Omron CX-Programmer project НовыйПроект (CX-Programmer 9.61)

# PLC НовыйПЛК1: CP1E N30

## Global symbols (name address type ; comment)
0.00 BOOL  ; Pulsador 00. Control valvula 00, easy box 1.
0.01 BOOL  ; Pulsadoe 01_control valvula 01. Easy box 2.
0.02 BOOL  ; Pulsador 02, activa valvula 02 y bomba B00_B01 en alternancia.
0.03 BOOL  ; Pulsador03, activa valvula 03.
0.04 BOOL  ; Pulsador 04, activa valvula 04 y G.Presion B00_B01.
0.05 BOOL  ; Pulsador05, activa valvula 05 y G.presion B00_B01.
100.00 BOOL  ; Valvula V00
100.01 BOOL  ; Valvula V01
100.02 BOOL  ; Valvula V02.
100.03 BOOL  ; Valvula V03.
100.04 BOOL  ; Valvula V04.
100.05 BOOL  ; Valvula V05.
101.00 BOOL  ; Bomba B00.
101.01 BOOL  ; Bomba B01.
101.02 BOOL  ; Bomba Filtracion f01
101.03 BOOL  ; Bomba Filtracion f02
1.00 BOOL  ; Guardamotor B00.
1.01 BOOL  ; Guardamotor B01.
1.02 BOOL  ; Guardamotor filtraciуn.
1.03 BOOL  ; Reloj_termostato filtracion.
D0 CHANNEL  ; D.M Valor activar bomba B00
D1 CHANNEL  ; D.M Valor temporizacion B00
D10 CHANNEL  ; D.M Valor activar bomba B01
D11 CHANNEL  ; D.M valor temporizacion B01
T000 BOOL  ; Retardo V02 arranque bomba B00_B01,
T001 BOOL  ; Retardo V02 arranque bomba B00_B01,
T002 BOOL  ; Retardo V02 arranque bomba B00_B01,
T003 BOOL  ; Retardo V03 arranque bomba B00_B01,
T004 BOOL  ; Retardo V04 arranque bomba B00_B01,
T005 BOOL  ; Retardo V05 arranque bomba B00_B01,
W0.00 BOOL  ; Trabajo pulsador 00_valvula 00
W0.01 BOOL  ; Trabajo pulsador 00_valvula00
W0.02 BOOL  ; Salida Virtual valvula00
W0.05 BOOL  ; Trabajo Pulsador01_valvula01
W0.06 BOOL  ; Trabajo pulsador01_valvula01.
W0.07 BOOL  ; Salida Virtual valvula 01.
W0.10 BOOL  ; Trabajo pulsador02_valvula02
W0.11 BOOL  ; Trabajo pulsador02_valvula02
W0.12 BOOL  ; Salida virtual valvula02
W100 CHANNEL  ; Temporal valor bomba B00
W100.00 BOOL  ; Salida virtual Bomba B00
W100.01 BOOL  ; Salida virtual bomba B01
W100.10 BOOL  ; Salida virtual filtraciуn.
W101 CHANNEL  ; Temporal bomba B01
W101.01 BOOL  ; Virtual bomba B01
W1.00 BOOL  ; Trabajo pulsador03_valvula03.
W1.01 BOOL  ; Trabajo pulsador03_valvula03
W1.02 BOOL  ; Salida virtual valvula03
W1.05 BOOL  ; Trabajo pulsador04_valvula04
W1.06 BOOL  ; Trabajo pulsador04_valvula04
W1.07 BOOL  ; Salida virtual valvula04
W1.10 BOOL  ; Trabajo pulsador 05_valvula05
W1.11 BOOL  ; Trabajo pulsador05_valvula05
W1.12 BOOL  ; Salida virtual valvula05
W20.00 BOOL  ; Salida virtual valvula 00
W20.01 BOOL  ; Salida virtual valvula 01
W20.02 BOOL  ; Salida virtual valvula 02
W20.03 BOOL  ; Salida virtual valvula 03
W20.04 BOOL  ; Salida virtual valvula 04
W20.05 BOOL  ; Salida virtual valvula 05
W20.10 BOOL  ; Виртуальна переменная для ыключения насоса 01
W20.11 BOOL  ; Виртуальна переменная для ыключения насоса 02
W30.00 BOOL  ; Salida virtual valvula02
W30.02 BOOL  ; Seсal V02 arranque B00_B01.
W50 CHANNEL  ; Registro incremento temporizacion alternancia

## Program NuevoPrograma1 (cyclic task 0)
Local symbols
do CHANNEL

### Section Enclavamiento_pulsadores

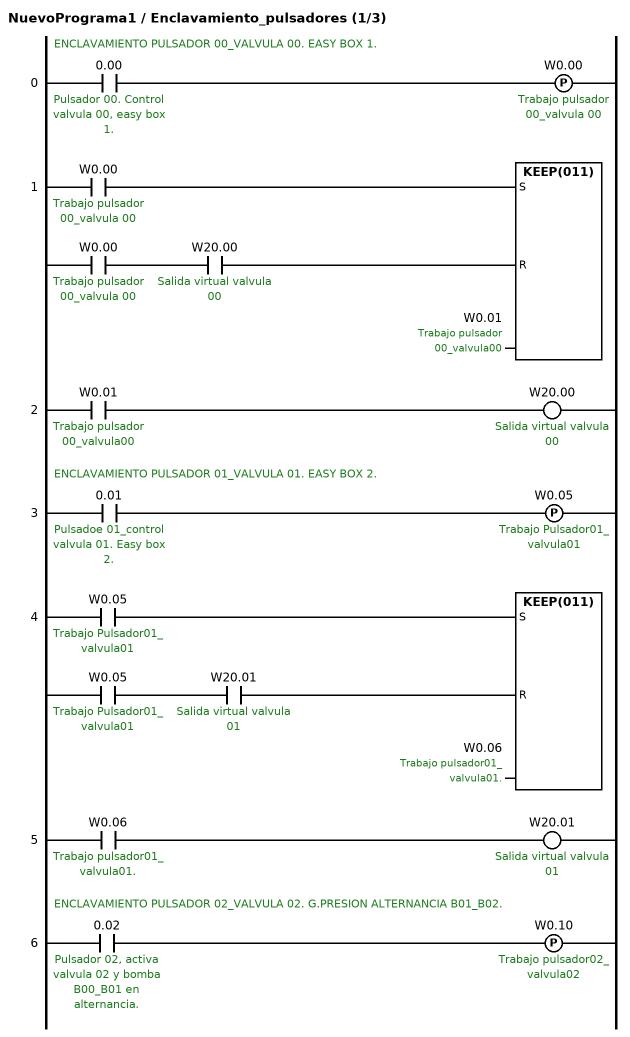
; rung 0: ENCLAVAMIENTO PULSADOR 00_VALVULA 00. EASY BOX 1.
LD 0.00  ; Pulsador 00. Control valvula 00, easy box 1.
DIFU(013) W0.00  ; Trabajo pulsador 00_valvula 00
; rung 1
LD W0.00  ; Trabajo pulsador 00_valvula 00
LD W0.00  ; Trabajo pulsador 00_valvula 00
AND W20.00  ; Salida virtual valvula 00
KEEP(011) W0.01  ; Trabajo pulsador 00_valvula00
; rung 2
LD W0.01  ; Trabajo pulsador 00_valvula00
OUT W20.00  ; Salida virtual valvula 00
; rung 3: ENCLAVAMIENTO PULSADOR 01_VALVULA 01. EASY BOX 2.
LD 0.01  ; Pulsadoe 01_control valvula 01. Easy box 2.
DIFU(013) W0.05  ; Trabajo Pulsador01_valvula01
; rung 4
LD W0.05  ; Trabajo Pulsador01_valvula01
LD W0.05  ; Trabajo Pulsador01_valvula01
AND W20.01  ; Salida virtual valvula 01
KEEP(011) W0.06  ; Trabajo pulsador01_valvula01.
; rung 5
LD W0.06  ; Trabajo pulsador01_valvula01.
OUT W20.01  ; Salida virtual valvula 01
; rung 6: ENCLAVAMIENTO PULSADOR 02_VALVULA 02. G.PRESION ALTERNANCIA B01_B02.
LD 0.02  ; Pulsador 02, activa valvula 02 y bomba B00_B01 en alternancia.
DIFU(013) W0.10  ; Trabajo pulsador02_valvula02

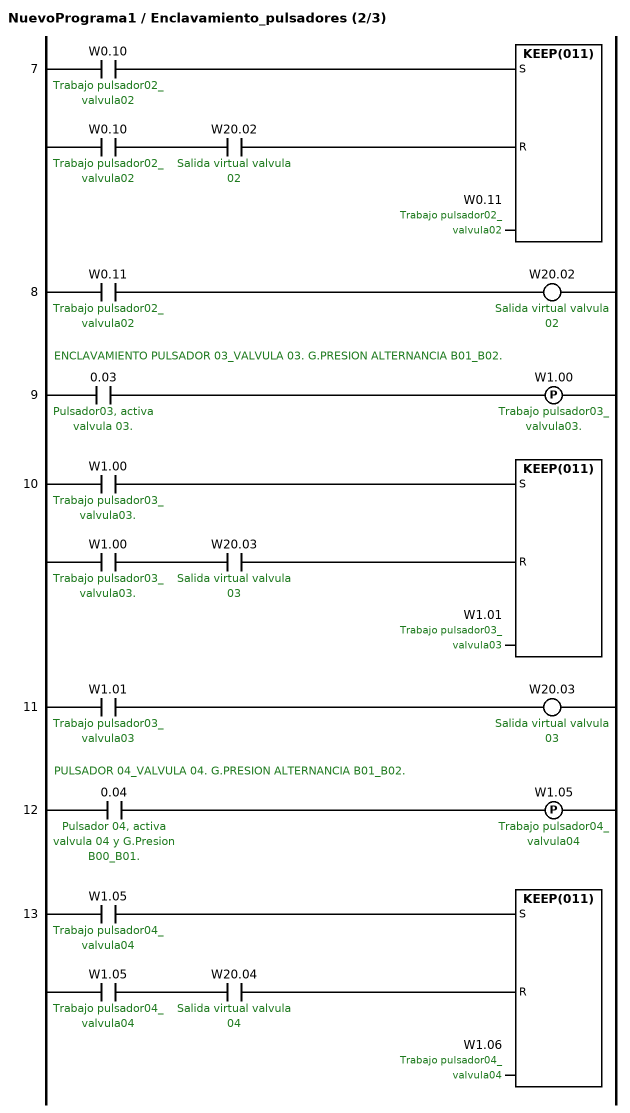
; rung 7
LD W0.10  ; Trabajo pulsador02_valvula02
LD W0.10  ; Trabajo pulsador02_valvula02
AND W20.02  ; Salida virtual valvula 02
KEEP(011) W0.11  ; Trabajo pulsador02_valvula02
; rung 8
LD W0.11  ; Trabajo pulsador02_valvula02
OUT W20.02  ; Salida virtual valvula 02
; rung 9: ENCLAVAMIENTO PULSADOR 03_VALVULA 03. G.PRESION ALTERNANCIA B01_B02.
LD 0.03  ; Pulsador03, activa valvula 03.
DIFU(013) W1.00  ; Trabajo pulsador03_valvula03.
; rung 10
LD W1.00  ; Trabajo pulsador03_valvula03.
LD W1.00  ; Trabajo pulsador03_valvula03.
AND W20.03  ; Salida virtual valvula 03
KEEP(011) W1.01  ; Trabajo pulsador03_valvula03
; rung 11
LD W1.01  ; Trabajo pulsador03_valvula03
OUT W20.03  ; Salida virtual valvula 03
; rung 12: PULSADOR 04_VALVULA 04. G.PRESION ALTERNANCIA B01_B02.
LD 0.04  ; Pulsador 04, activa valvula 04 y G.Presion B00_B01.
DIFU(013) W1.05  ; Trabajo pulsador04_valvula04
; rung 13
LD W1.05  ; Trabajo pulsador04_valvula04
LD W1.05  ; Trabajo pulsador04_valvula04
AND W20.04  ; Salida virtual valvula 04
KEEP(011) W1.06  ; Trabajo pulsador04_valvula04

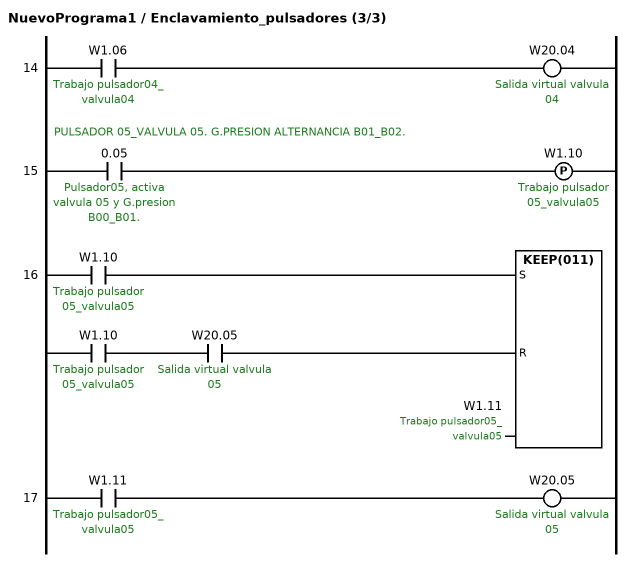
; rung 14
LD W1.06  ; Trabajo pulsador04_valvula04
OUT W20.04  ; Salida virtual valvula 04
; rung 15: PULSADOR 05_VALVULA 05. G.PRESION ALTERNANCIA B01_B02.
LD 0.05  ; Pulsador05, activa valvula 05 y G.presion B00_B01.
DIFU(013) W1.10  ; Trabajo pulsador 05_valvula05
; rung 16
LD W1.10  ; Trabajo pulsador 05_valvula05
LD W1.10  ; Trabajo pulsador 05_valvula05
AND W20.05  ; Salida virtual valvula 05
KEEP(011) W1.11  ; Trabajo pulsador05_valvula05
; rung 17
LD W1.11  ; Trabajo pulsador05_valvula05
OUT W20.05  ; Salida virtual valvula 05

### Section Alternancia_bombas_B00_B01

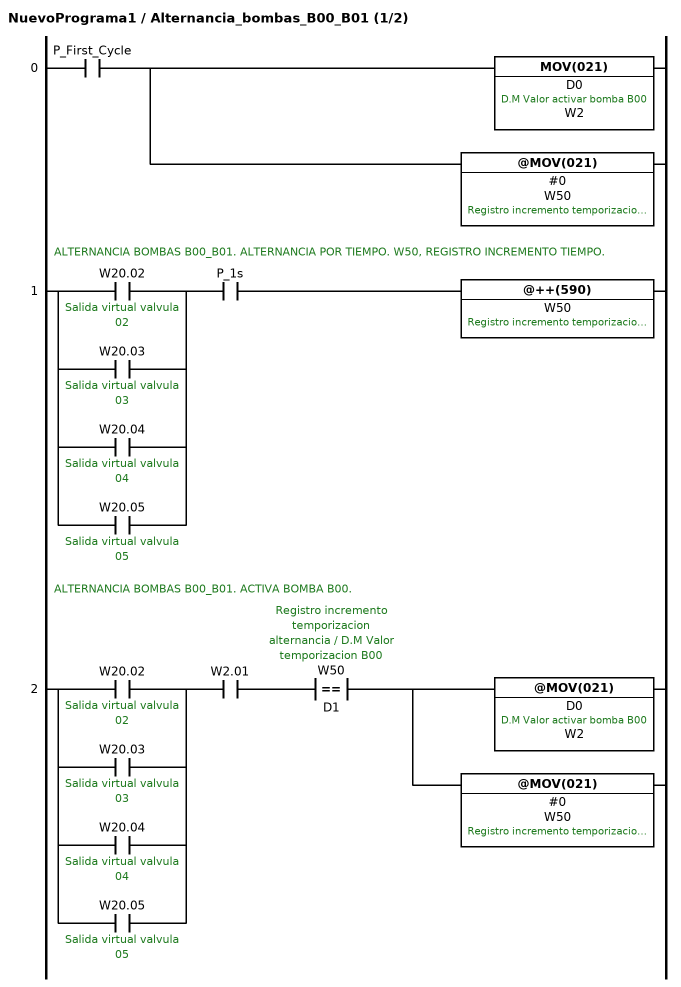
; rung 0
LD P_First_Cycle
MOV(021) D0 W2  ; D.M Valor activar bomba B00
@MOV(021) #0 W50  ; Registro incremento temporizacion alternancia
; rung 1: ALTERNANCIA BOMBAS B00_B01. ALTERNANCIA POR TIEMPO. W50, REGISTRO INCREMENTO TIEMPO.
LD W20.02  ; Salida virtual valvula 02
OR W20.03  ; Salida virtual valvula 03
OR W20.04  ; Salida virtual valvula 04
OR W20.05  ; Salida virtual valvula 05
AND P_1s
@++(590) W50  ; Registro incremento temporizacion alternancia
; rung 2: ALTERNANCIA BOMBAS B00_B01. ACTIVA BOMBA B00.
LD W20.02  ; Salida virtual valvula 02
OR W20.03  ; Salida virtual valvula 03
OR W20.04  ; Salida virtual valvula 04
OR W20.05  ; Salida virtual valvula 05
AND W2.01
AND=(300) W50 D1  ; Registro incremento temporizacion alternancia, D.M Valor temporizacion B00
@MOV(021) D0 W2  ; D.M Valor activar bomba B00
@MOV(021) #0 W50  ; Registro incremento temporizacion alternancia

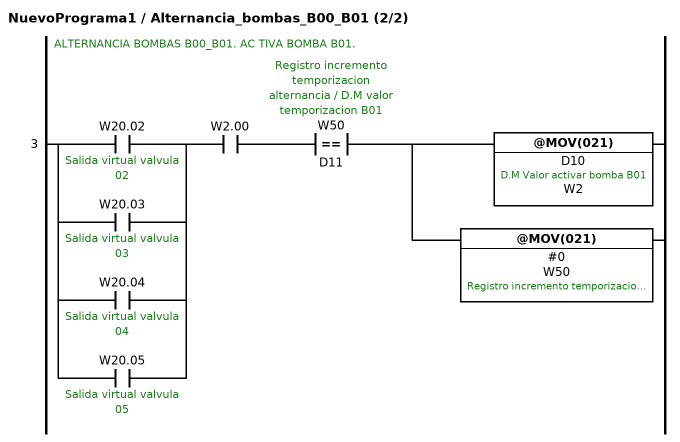
; rung 3: ALTERNANCIA BOMBAS B00_B01. AC TIVA BOMBA B01.
LD W20.02  ; Salida virtual valvula 02
OR W20.03  ; Salida virtual valvula 03
OR W20.04  ; Salida virtual valvula 04
OR W20.05  ; Salida virtual valvula 05
AND W2.00
AND=(300) W50 D11  ; Registro incremento temporizacion alternancia, D.M valor temporizacion B01
@MOV(021) D10 W2  ; D.M Valor activar bomba B01
@MOV(021) #0 W50  ; Registro incremento temporizacion alternancia

### Section Retardos_arranque_bombas00_01

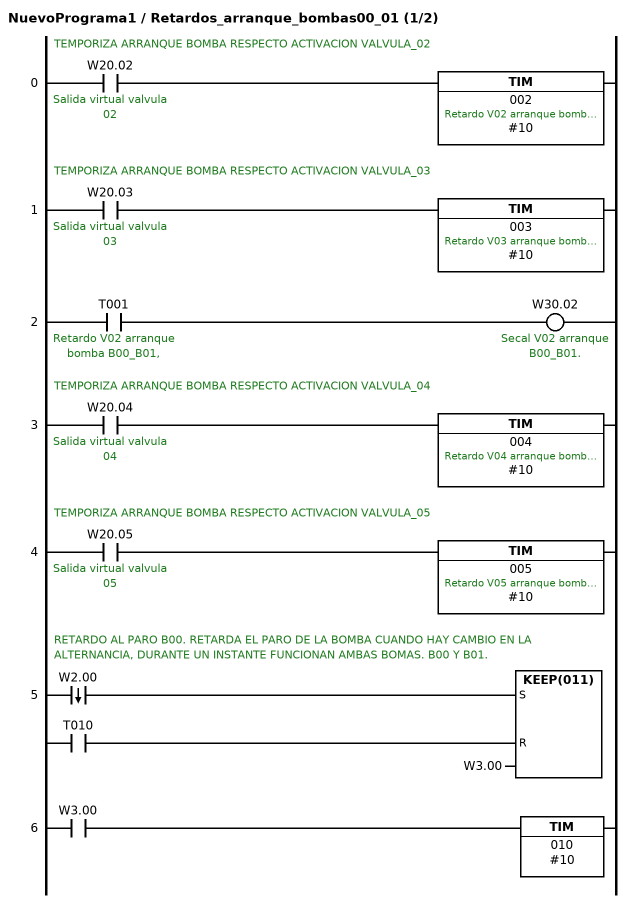
; rung 0: TEMPORIZA ARRANQUE BOMBA RESPECTO ACTIVACION VALVULA_02
LD W20.02  ; Salida virtual valvula 02
TIM 002 #10  ; Retardo V02 arranque bomba B00_B01,
; rung 1: TEMPORIZA ARRANQUE BOMBA RESPECTO ACTIVACION VALVULA_03
LD W20.03  ; Salida virtual valvula 03
TIM 003 #10  ; Retardo V03 arranque bomba B00_B01,
; rung 2
LD T001  ; Retardo V02 arranque bomba B00_B01,
OUT W30.02  ; Seсal V02 arranque B00_B01.
; rung 3: TEMPORIZA ARRANQUE BOMBA RESPECTO ACTIVACION VALVULA_04
LD W20.04  ; Salida virtual valvula 04
TIM 004 #10  ; Retardo V04 arranque bomba B00_B01,
; rung 4: TEMPORIZA ARRANQUE BOMBA RESPECTO ACTIVACION VALVULA_05
LD W20.05  ; Salida virtual valvula 05
TIM 005 #10  ; Retardo V05 arranque bomba B00_B01,
; rung 5: RETARDO AL PARO B00. RETARDA EL PARO DE LA BOMBA CUANDO HAY CAMBIO EN LA ALTERNANCIA, DURANTE UN INSTANTE FUNCIONAN AMBAS BOMAS. B00 Y B01.
%LD W2.00
LD T010
KEEP(011) W3.00
; rung 6
LD W3.00
TIM 010 #10

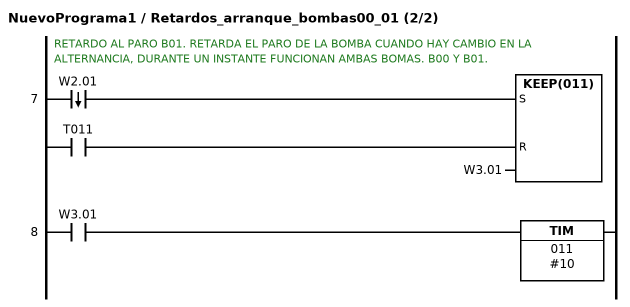
; rung 7: RETARDO AL PARO B01. RETARDA EL PARO DE LA BOMBA CUANDO HAY CAMBIO EN LA ALTERNANCIA, DURANTE UN INSTANTE FUNCIONAN AMBAS BOMAS. B00 Y B01.
%LD W2.01
LD T011
KEEP(011) W3.01
; rung 8
LD W3.01
TIM 011 #10

### Section Salidas

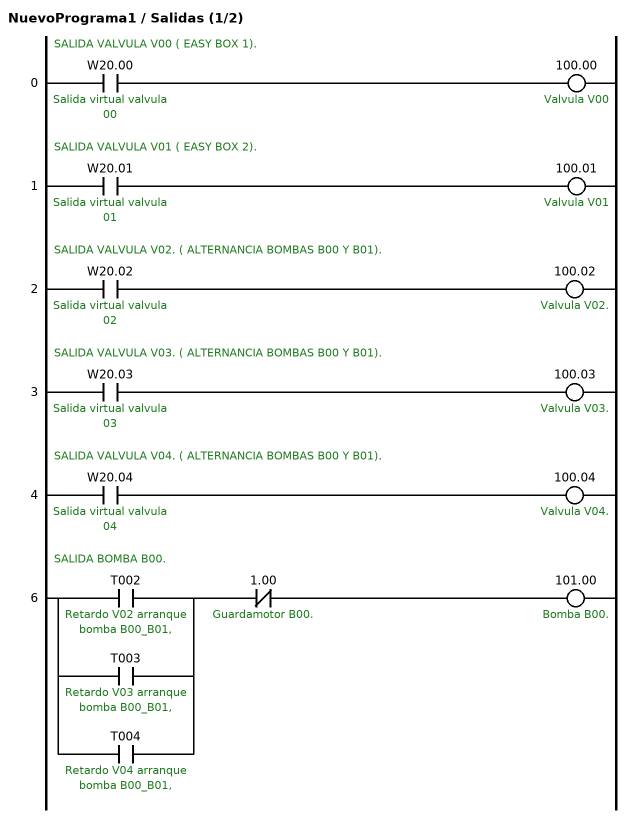
; rung 0: SALIDA VALVULA V00 ( EASY BOX 1).
LD W20.00  ; Salida virtual valvula 00
OUT 100.00  ; Valvula V00
; rung 1: SALIDA VALVULA V01 ( EASY BOX 2).
LD W20.01  ; Salida virtual valvula 01
OUT 100.01  ; Valvula V01
; rung 2: SALIDA VALVULA V02. ( ALTERNANCIA BOMBAS B00 Y B01).
LD W20.02  ; Salida virtual valvula 02
OUT 100.02  ; Valvula V02.
; rung 3: SALIDA VALVULA V03. ( ALTERNANCIA BOMBAS B00 Y B01).
LD W20.03  ; Salida virtual valvula 03
OUT 100.03  ; Valvula V03.
; rung 4: SALIDA VALVULA V04. ( ALTERNANCIA BOMBAS B00 Y B01).
LD W20.04  ; Salida virtual valvula 04
OUT 100.04  ; Valvula V04.
; rung 5: SALIDA VALVULA V05. ( ALTERNANCIA BOMBAS B00 Y B01).
; rung 6: SALIDA BOMBA B00.
LD T002  ; Retardo V02 arranque bomba B00_B01,
OR T003  ; Retardo V03 arranque bomba B00_B01,
OR T004  ; Retardo V04 arranque bomba B00_B01,
ANDNOT 1.00  ; Guardamotor B00.
OUT 101.00  ; Bomba B00.

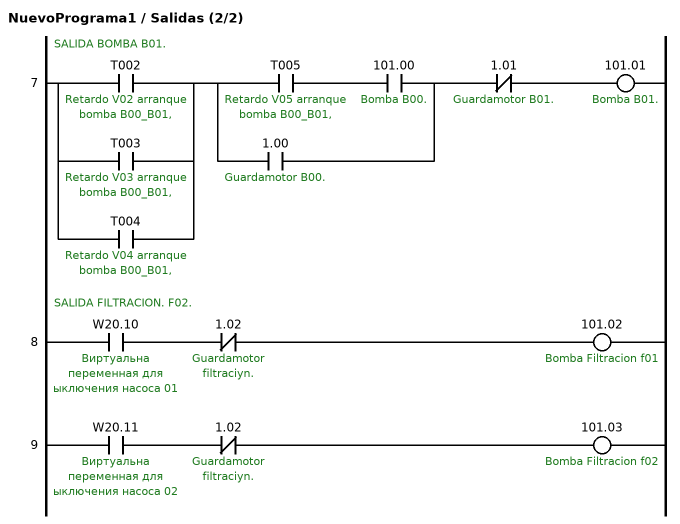
; rung 7: SALIDA BOMBA B01.
LD T002  ; Retardo V02 arranque bomba B00_B01,
OR T003  ; Retardo V03 arranque bomba B00_B01,
OR T004  ; Retardo V04 arranque bomba B00_B01,
LD T005  ; Retardo V05 arranque bomba B00_B01,
AND 101.00  ; Bomba B00.
OR 1.00  ; Guardamotor B00.
ANDLD
ANDNOT 1.01  ; Guardamotor B01.
OUT 101.01  ; Bomba B01.
; rung 8: SALIDA FILTRACION. F02.
LD W20.10  ; Виртуальна переменная для ыключения насоса 01
ANDNOT 1.02  ; Guardamotor filtraciуn.
OUT 101.02  ; Bomba Filtracion f01
; rung 9
LD W20.11  ; Виртуальна переменная для ыключения насоса 02
ANDNOT 1.02  ; Guardamotor filtraciуn.
OUT 101.03  ; Bomba Filtracion f02

### Section DoseBombaFiltrado

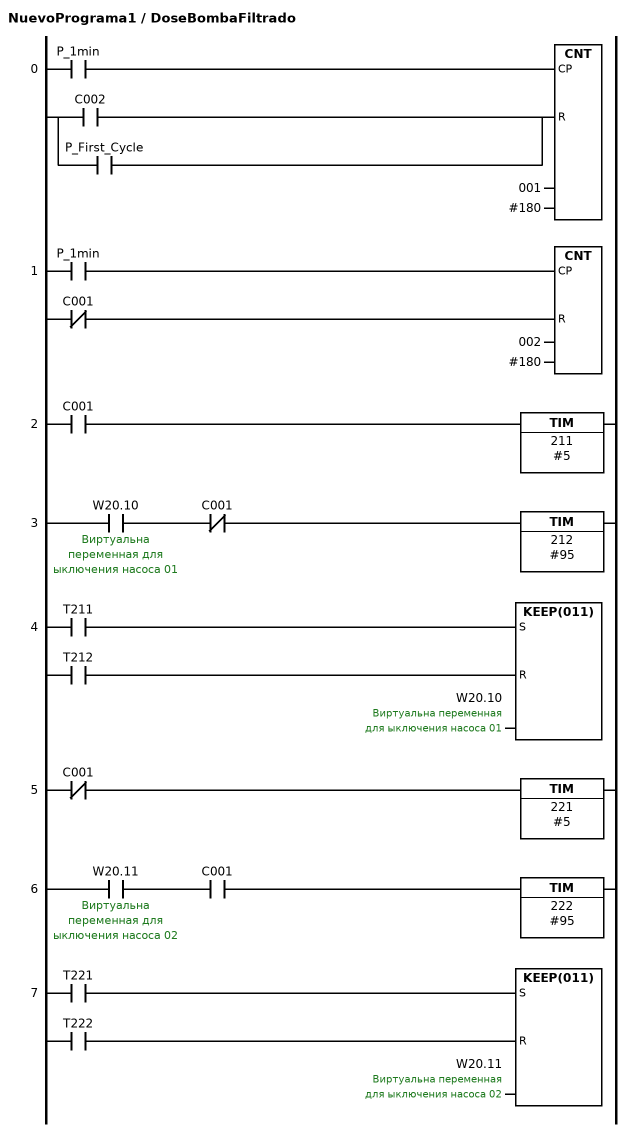
; rung 0
LD P_1min
LD C002
OR P_First_Cycle
CNT 001 #180
; rung 1
LD P_1min
LDNOT C001
CNT 002 #180
; rung 2
LD C001
TIM 211 #5
; rung 3
LD W20.10  ; Виртуальна переменная для ыключения насоса 01
ANDNOT C001
TIM 212 #95
; rung 4
LD T211
LD T212
KEEP(011) W20.10  ; Виртуальна переменная для ыключения насоса 01
; rung 5
LDNOT C001
TIM 221 #5
; rung 6
LD W20.11  ; Виртуальна переменная для ыключения насоса 02
AND C001
TIM 222 #95
; rung 7
LD T221
LD T222
KEEP(011) W20.11  ; Виртуальна переменная для ыключения насоса 02

### Section END
; rung 0
END(001)